Universal Robots PolyScope program: programa1.urp

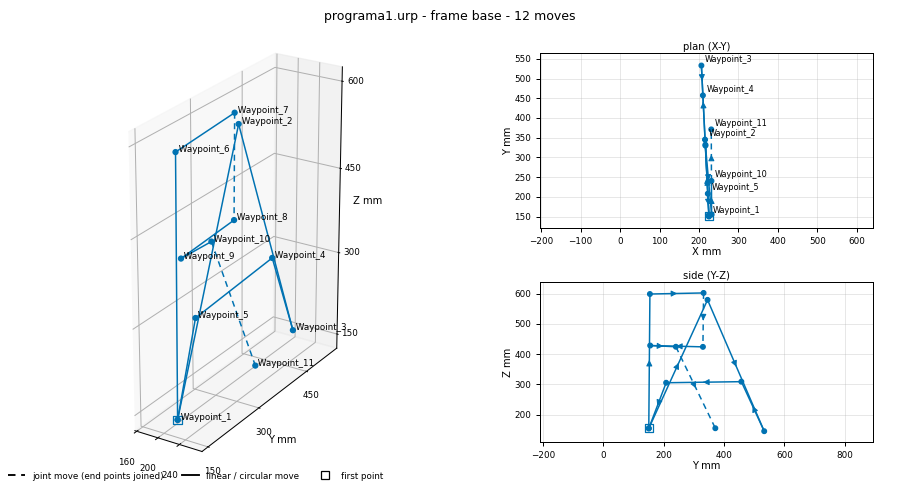
[picture p0: tool path of programa1.urp in frame base, 12 of 12 moves have a stored position in this frame; points joined in program order, loops and branches not executed]
Program programa1 (installation=default directory=/ursim/programs createdIn=5.26.1 lastSavedIn=5.26.1 robotSerialNumber=20195599999)
Calibrated DH parameters: a=[0, -0.425, -0.3922, 0, 0, 0]; d=[0.1625, 0, 0, 0.1333, 0.0997, 0.0996]; alpha=[1.570796, 0, 0, 1.570796, -1.570796, 0]; deltaTheta=[0, 0, 0, 0, 0, 0]
InitVariablesNode
Robot Program (runOnlyOnce=false)
  Popup Message (haltProgram=false message=realizando la letra 'A' de (Andres) inputType=Text)
  MoveL speed 250 mm/s, acceleration 1200 mm/s^2 (useActiveTCP=true optimoveEnabled=false optiMoveSpeed=0.3 optiMoveAcceleration=0.09) feature=Base
    Waypoint Waypoint_1: TCP in base x=225.191 y=150.784 z=154.325 mm, rx=1.6237 ry=0.8752 rz=1.5468 rad; joints [92.857, -76.709, -158.634, -111.037, 5.59, 17.217] deg; TCP offset x=0 y=0 z=0 mm, rx=0 ry=0 rz=0 rad
  MoveL speed 250 mm/s, acceleration 1200 mm/s^2 (useActiveTCP=true optimoveEnabled=false optiMoveSpeed=0.3 optiMoveAcceleration=0.09) feature=Base
    Waypoint Waypoint_2: TCP in base x=215.251 y=345.315 z=579.769 mm, rx=-2.1781 ry=0.2673 rz=-1.9189 rad; joints [92.857, -68.447, -106.499, -95.469, 6.828, 17.217] deg; TCP offset x=0 y=0 z=0 mm, rx=0 ry=0 rz=0 rad
  MoveL speed 250 mm/s, acceleration 1200 mm/s^2 (useActiveTCP=true optimoveEnabled=false optiMoveSpeed=0.3 optiMoveAcceleration=0.09) feature=Base
    Waypoint Waypoint_3: TCP in base x=206.121 y=532.955 z=144.97 mm, rx=1.7399 ry=0.7748 rz=1.6447 rad; joints [92.857, -121.527, -104.869, -111.037, 5.59, 17.217] deg; TCP offset x=0 y=0 z=0 mm, rx=0 ry=0 rz=0 rad
  MoveL speed 250 mm/s, acceleration 1200 mm/s^2 (useActiveTCP=true optimoveEnabled=false optiMoveSpeed=0.3 optiMoveAcceleration=0.09) feature=Base
    Waypoint Waypoint_4: TCP in base x=209.898 y=457.27 z=308.956 mm, rx=1.9532 ry=0.5586 rz=1.8216 rad; joints [92.857, -96.573, -112.852, -111.037, 5.59, 17.217] deg; TCP offset x=0 y=0 z=0 mm, rx=0 ry=0 rz=0 rad
  MoveL speed 250 mm/s, acceleration 1200 mm/s^2 (useActiveTCP=true optimoveEnabled=false optiMoveSpeed=0.3 optiMoveAcceleration=0.09) feature=Base
    Waypoint Waypoint_5: TCP in base x=222.323 y=208.27 z=305.402 mm, rx=2.0652 ry=0.4248 rz=1.913 rad; joints [92.857, -55.616, -144.505, -111.037, 5.59, 17.217] deg; TCP offset x=0 y=0 z=0 mm, rx=0 ry=0 rz=0 rad
  Popup Message (haltProgram=false message=realizando la letra 'R' de (Rivera) inputType=Text)
  MoveL speed 250 mm/s, acceleration 1200 mm/s^2 (useActiveTCP=true optimoveEnabled=false optiMoveSpeed=0.3 optiMoveAcceleration=0.09) feature=Base
    Waypoint Waypoint_1: TCP in base x=225.191 y=150.784 z=154.325 mm, rx=1.6237 ry=0.8752 rz=1.5468 rad; joints [92.857, -76.709, -158.634, -111.037, 5.59, 17.217] deg; TCP offset x=0 y=0 z=0 mm, rx=0 ry=0 rz=0 rad
  MoveL speed 250 mm/s, acceleration 1200 mm/s^2 (useActiveTCP=true optimoveEnabled=false optiMoveSpeed=0.3 optiMoveAcceleration=0.09) feature=Base
    Waypoint Waypoint_6: TCP in base x=225.132 y=154.508 z=599.155 mm, rx=1.8358 ry=0.6852 rz=1.7443 rad; joints [92.857, -54.267, -98.141, -176.921, 4.788, 17.217] deg; TCP offset x=0 y=0 z=0 mm, rx=0 ry=0 rz=0 rad
  MoveL speed 250 mm/s, acceleration 1200 mm/s^2 (useActiveTCP=true optimoveEnabled=false optiMoveSpeed=0.3 optiMoveAcceleration=0.09) feature=Base
    Waypoint Waypoint_7: TCP in base x=216.266 y=332.184 z=602.718 mm, rx=1.7102 ry=0.8062 rz=1.6375 rad; joints [92.857, -79.116, -83.215, -176.921, 4.788, 17.217] deg; TCP offset x=0 y=0 z=0 mm, rx=0 ry=0 rz=0 rad
  MoveJ speed 60 deg/s, acceleration 80 deg/s^2 (useActiveTCP=true optimoveEnabled=false optiMoveSpeed=0.3 optiMoveAcceleration=0.09) feature=Base
    Waypoint Waypoint_8: TCP in base x=216.374 y=330.02 z=424.208 mm, rx=1.3573 ry=1.0775 rz=1.3324 rad; joints [92.857, -83.287, -105.824, -176.921, 4.788, 17.217] deg; TCP offset x=0 y=0 z=0 mm, rx=0 ry=0 rz=0 rad
  MoveL speed 250 mm/s, acceleration 1200 mm/s^2 (useActiveTCP=true optimoveEnabled=false optiMoveSpeed=0.3 optiMoveAcceleration=0.09) feature=Base
    Waypoint Waypoint_9: TCP in base x=231.945 y=155.459 z=428.607 mm, rx=1.5192 ry=0.9332 rz=1.4298 rad; joints [90.225, -55.937, -122.007, -176.921, 4.788, 17.217] deg; TCP offset x=0 y=0 z=0 mm, rx=0 ry=0 rz=0 rad
  MoveL speed 250 mm/s, acceleration 1200 mm/s^2 (useActiveTCP=true optimoveEnabled=false optiMoveSpeed=0.3 optiMoveAcceleration=0.09) feature=Base
    Waypoint Waypoint_10: TCP in base x=231.611 y=240.495 z=424.567 mm, rx=1.4147 ry=1.0119 rz=1.3355 rad; joints [90.225, -71.187, -114.826, -176.921, 4.788, 17.217] deg; TCP offset x=0 y=0 z=0 mm, rx=0 ry=0 rz=0 rad
  MoveJ speed 60 deg/s, acceleration 80 deg/s^2 (useActiveTCP=true optimoveEnabled=false optiMoveSpeed=0.3 optiMoveAcceleration=0.09) feature=Base
    Waypoint Waypoint_11: TCP in base x=231.099 y=371.109 z=154.777 mm, rx=0.7747 ry=1.3473 rz=0.7542 rad; joints [90.225, -120.953, -112.476, -176.921, 4.788, 17.217] deg; TCP offset x=0 y=0 z=0 mm, rx=0 ry=0 rz=0 rad
